Fanuc KAREL source: kc00002.KL

-- PROVISIONAL review KL for V940-1; original PC SHA256 b0da157ce530dedff3ae6a9dc1ab8f78b6eb60ac831736d9f0c273122a89741e
-- Incomplete behavior may be omitted. Consult companion uncertainty JSON. Do not deploy.
PROGRAM KC00002
%NOLOCKGROUP
BEGIN
  -- V9_ZERO_TABLE_METADATA_HINT layout=0002_ascii; no indexed target words; source/name/runtime held
  -- UNRESOLVED_PC offsets 5-33; opcodes 27,22,22,22,22,31
  -- UNRESOLVED_PC offsets 38-42; opcodes 7F
END KC00002
